// TwinCAT 3 PLC project TcCommando
// Title: TcCommando
// Company: Loupe
// Author: Loupe
// ProjectVersion: 0.0.1
// ProgramVersion: 3.1.4024.0
// libraries:
//   Tc2_Standard, * (Beckhoff Automation GmbH)
//   Tc2_System, * (Beckhoff Automation GmbH)
//   Tc3_Module, * (Beckhoff Automation GmbH)
//   TcPluginFramework, * (Loupe)
// project tree:
//   PLCOpen/DUT/ PLCOpenCallInternal.TcDUT, PLCOpenCallState.TcTLEO, PLCOpenCommandInternal.TcDUT (not stored), PLCOpenStatusBase.TcTLEO (not stored)
//   PLCOpen/Interfaces/ IPLCOpenBase.TcIO (not stored), IPLCOpenCall.TcIO, IPLCOpenCommand.TcIO (not stored), IPLCOpenGroup.TcIO
//   PLCOpen/POU/ PLCOpenCall.TcPOU, PLCOpenCallGroup.TcPOU (not stored), PLCOpenCallGroupType.TcDUT, PLCOpenCommand.TcPOU (not stored), PLCOpenCommandGroup.TcPOU, PLCOpenNullRemote.TcPOU (not stored)
//   / PlcTask.TcTTO
//   POUs/ MAIN.TcPOU (not stored)
// real-time tasks:
//   TASK PlcTask: cycle T#10ms, priority 20, ADS port 350

CONFIGURATION TcCommando
    RESOURCE PLC ON TwinCAT3
        TASK PlcTask(INTERVAL := T#10ms, PRIORITY := 20);
        PROGRAM MAIN WITH PlcTask : MAIN;
    END_RESOURCE
END_CONFIGURATION

// ---- PLCOpen/DUT/PLCOpenCallInternal.TcDUT
TYPE PLCOpenCallInternal :
STRUCT
	_state : PLCOpenCallState;
	_Command: IPLCOpenCommand;
	_abort: BOOL;
	_execute: BOOL;
	_break:BOOL;
	_RemoteStatus: PLCOPENSTATUSBASE;
	_self :IPLCOpenCall;
END_STRUCT
END_TYPE

// ---- PLCOpen/DUT/PLCOpenCallState.TcTLEO
{attribute 'qualified_only'}
{attribute 'strict'}
TYPE PLCOpenCallState :
(
	ATN_PLCOPEN_FUB_IDLE := 0,
	ATN_PLCOPEN_FUB_NEW_COMMAND,
	ATN_PLCOPEN_FUB_ABORTED,
	ATN_PLCOPEN_FUB_ABORT_OLD,
	ATN_PLCOPEN_FUB_STATUS,
	ATN_PLCOPEN_FUB_WRITE_PAR,
	ATN_PLCOPEN_FUB_SET_COMMAND,
	ATN_PLCOPEN_FUB_WORKING,
	ATN_PLCOPEN_FUB_CLEANUP,
	ATN_PLCOPEN_FUB_DONE
);
END_TYPE

// ---- PLCOpen/POU/PLCOpenCallGroupType.TcDUT
TYPE PLCOpenCallGroupType :
STRUCT
	_startStep : ENUM;  //The step when doStep was called
	_currentStep :ENUM;
	_lastRequestNumber : DINT;
	_onEntry : BOOL;
	_onExit : BOOL;
	_isDone : BOOL;
	_isAbort : BOOL;
	_isError : BOOL;
	_statusChecked : BOOL;
	_numberActiveCommands : INT;
	_commands : ARRAY[0..19] OF PLCOpenCall;
	_syncAbort : BOOL;
	_syncError : BOOL;
	_syncDone : BOOL;
END_STRUCT
END_TYPE

// ---- PLCOpen/Interfaces/IPLCOpenCall.TcIO
INTERFACE IPLCOpenCall

METHOD Aborted : BOOL
VAR_INPUT
END_VAR
END_METHOD

METHOD Errored : BOOL
VAR_INPUT
	ID : INT;
END_VAR
END_METHOD

METHOD Finished : BOOL
VAR_INPUT
END_VAR
END_METHOD

METHOD Start : BOOL
VAR_INPUT
	Command : IPLCOpenCommand;	
END_VAR
END_METHOD

END_INTERFACE

// ---- PLCOpen/Interfaces/IPLCOpenGroup.TcIO
INTERFACE IPLCOpenGroup

METHOD AbortPreviousCommands : BOOL
VAR_INPUT
	newCommand : IPLCOpenCommand;
END_VAR
END_METHOD

END_INTERFACE

// ---- PLCOpen/POU/PLCOpenCall.TcPOU
FUNCTION_BLOCK PLCOpenCall IMPLEMENTS IPLCOpenCall 
VAR_INPUT
	Execute : BOOL;
	Command : IPLCOpenCommand;
	Fallback: PLCOPENSTATUSBASE;
END_VAR
VAR_OUTPUT
	Status: PLCOPENSTATUSBASE;
	Busy : BOOL;
	Done : BOOL;
	Error : BOOL;
	CommandAborted : BOOL;
END_VAR
VAR
	i_PLCOpenCallInternal : PLCOpenCallInternal;
END_VAR

Call();

METHOD Aborted : BOOL
i_PLCOpenCallInternal._abort := true;
END_METHOD

METHOD Call : BOOL
VAR
	_break : BOOL;
END_VAR
	//Capture edges
	IF NOT Execute THEN
		i_PLCOpenCallInternal._execute := FALSE;
	END_IF

	//Start a new command on edge
	IF( Execute AND NOT i_PLCOpenCallInternal._execute)THEN
		i_PLCOpenCallInternal._execute := TRUE;
		i_PLCOpenCallInternal._state := PLCOpenCallState.ATN_PLCOPEN_FUB_NEW_COMMAND;
	END_IF
	
	//If we get aborted, handle it
	IF( i_PLCOpenCallInternal._abort )THEN
		i_PLCOpenCallInternal._abort := 0;
		i_PLCOpenCallInternal._state := PLCOpenCallState.ATN_PLCOPEN_FUB_ABORTED;
	END_IF

	i_PLCOpenCallInternal._self := THIS^;
	
	//We use a while not break so that we can do multiple passes at the state machine to do as much as possible in a single call	
	_break := FALSE;
	WHILE _break = FALSE DO
		CASE ( i_PLCOpenCallInternal._state ) OF
			//IDLE
			PLCOpenCallState.ATN_PLCOPEN_FUB_IDLE:
				Status := PLCOpenStatusBase.NOT_ENABLED;
				Busy := FALSE;
				Done := FALSE;
				Error := FALSE;
				CommandAborted := FALSE;
				_break := TRUE;
				
			//Start a new command by getting it
			PLCOpenCallState.ATN_PLCOPEN_FUB_NEW_COMMAND:
				Status := PLCOpenStatusBase.BUSY;
				i_PLCOpenCallInternal._RemoteStatus := PLCOpenStatusBase.BUSY;
				Busy := TRUE;
				Done := FALSE;
				Error := FALSE;
				CommandAborted := FALSE;			

				//If we are the current command:
				//1. we don't care about feedback
				//2. we don't want ourselves to get the abort
				//so remove this fub before calling abort previous
				IF i_PLCOpenCallInternal._Command <> 0 THEN
					IF i_PLCOpenCallInternal._Command.Remote = i_PLCOpenCallInternal._self THEN
						i_PLCOpenCallInternal._Command.Remote := 0; 
					END_IF
				END_IF 

				//Get the new command
				i_PLCOpenCallInternal._command := Command;
	
				IF i_PLCOpenCallInternal._Command <> 0 THEN
					i_PLCOpenCallInternal._state := PLCOpenCallState.ATN_PLCOPEN_FUB_ABORT_OLD;
					//No break;
				ELSE
					i_PLCOpenCallInternal._state := PLCOpenCallState.ATN_PLCOPEN_FUB_WORKING;
					i_PLCOpenCallInternal._RemoteStatus := Fallback;				
					_break := TRUE;
				END_IF

				//No break;
			
			//Abort any commands that was active using the same PLCOpen state
			PLCOpenCallState.ATN_PLCOPEN_FUB_ABORT_OLD:
				//This will 
				i_PLCOpenCallInternal._Command.AbortPreviousCommands(i_PLCOpenCallInternal._Command);

				i_PLCOpenCallInternal._state := PLCOpenCallState.ATN_PLCOPEN_FUB_SET_COMMAND;
				//no break;
				
			//Start the command
			PLCOpenCallState.ATN_PLCOPEN_FUB_SET_COMMAND:
				i_PLCOpenCallInternal._Command.Execute := TRUE;			
				i_PLCOpenCallInternal._Command.Remote := THIS^;			
			
				Busy := TRUE;
				i_PLCOpenCallInternal._state := PLCOpenCallState.ATN_PLCOPEN_FUB_WORKING;
				// no break
	
			//Wait for the command to be finished
			PLCOpenCallState.ATN_PLCOPEN_FUB_WORKING:
				Busy := TRUE;
				//No Break
	
				IF( i_PLCOpenCallInternal._RemoteStatus <> PLCOpenStatusBase.BUSY AND i_PLCOpenCallInternal._RemoteStatus <> PLCOpenStatusBase.ENABLED_WAITING ) THEN
					Status := i_PLCOpenCallInternal._RemoteStatus;
					Busy := FALSE;
					IF( Status = 0 ) THEN
						Done := TRUE;
					
					ELSE
						Error := TRUE;		
					END_IF
					i_PLCOpenCallInternal._state := PLCOpenCallState.ATN_PLCOPEN_FUB_CLEANUP;
					//no break;
				ELSE 
					_break := TRUE;
				END_IF
			
			//cleanup
			PLCOpenCallState.ATN_PLCOPEN_FUB_CLEANUP:
				//Remove self from the source command
				IF i_PLCOpenCallInternal._Command <> 0 THEN
					i_PLCOpenCallInternal._Command.Remote := 0;			
					i_PLCOpenCallInternal._Command := 0;
				END_IF
					
				i_PLCOpenCallInternal._state := PLCOpenCallState.ATN_PLCOPEN_FUB_DONE;
				//Break to force at least 1 cycle with statuses
				_break := TRUE;

			//done
			PLCOpenCallState.ATN_PLCOPEN_FUB_DONE:
	
				IF( NOT Execute )THEN
					i_PLCOpenCallInternal._state := PLCOpenCallState.ATN_PLCOPEN_FUB_IDLE;
					Status := PLCOpenStatusBase.NOT_ENABLED;
					Busy := FALSE;
					Done := FALSE;
					Error := FALSE;
					CommandAborted := FALSE;				
				END_IF
				_break := TRUE;
	
			//aborted
			PLCOpenCallState.ATN_PLCOPEN_FUB_ABORTED:
				Status := PLCOpenStatusBase.ABORTED;
				Busy := FALSE;
				Done := FALSE;
				Error := FALSE;
				CommandAborted := TRUE;
				i_PLCOpenCallInternal._command := 0;
				i_PLCOpenCallInternal._state := PLCOpenCallState.ATN_PLCOPEN_FUB_DONE;
				_break := TRUE;
					
		END_CASE
	END_WHILE
END_METHOD

METHOD Clear : PLCOpenStatusBase
THIS^.Execute := FALSE;
THIS^.i_PLCOpenCallInternal._state := PLCOpenCallState.ATN_PLCOPEN_FUB_CLEANUP;
//One call to cleanup
THIS^.Call();
//Second call to clear
THIS^.Call();
END_METHOD

METHOD Errored : BOOL
VAR_INPUT
	ID : INT;
END_VAR
CASE ID OF
	//Any of these statuses are invalid to return as an error.
	//Override to error
	PLCOPENSTATUSBASE.BUSY,
	PLCOPENSTATUSBASE.ENABLED_WAITING,
	PLCOPENSTATUSBASE.ERR_OK:
		i_PLCOpenCallInternal._RemoteStatus := PLCOPENSTATUSBASE.ERROR;
ELSE
	//Any other status can be passed through
	i_PLCOpenCallInternal._RemoteStatus := ID;
END_CASE
END_METHOD

METHOD Exec : PLCOpenStatusBase
VAR_INPUT
	Command : IPLCOpenCommand;	
END_VAR
//Abort the previous command if it exists
IF THIS^.Command <> Command THEN
	Command.Execute := FALSE;
	THIS^.Call();
END_IF

THIS^.Command := Command;
THIS^.Execute := TRUE;
THIS^.Call();
Exec := THIS^.Status;
END_METHOD

METHOD Finished : BOOL
i_PLCOpenCallInternal._RemoteStatus := PLCOpenStatusBase.ERR_OK;
END_METHOD

METHOD Start : BOOL
VAR_INPUT
	Command : IPLCOpenCommand;	
END_VAR
THIS^.Exec(Command);
END_METHOD

END_FUNCTION_BLOCK

// ---- PLCOpen/POU/PLCOpenCommandGroup.TcPOU
{attribute 'call_after_init'}
FUNCTION_BLOCK PLCOpenCommandGroup IMPLEMENTS IPLCOpenGroup
VAR_INPUT
	commands : ARRAY[0..19] OF  IPLCOpenCommand;
END_VAR

METHOD AbortPreviousCommands : BOOL
VAR_INPUT
	newCommand : IPLCOpenCommand;
END_VAR

VAR
	i: INT;
END_VAR
FOR i:=0 TO 19 DO

	IF commands[i] <> 0 AND commands[i] <> newCommand THEN

		commands[i].Aborted();

	END_IF	

END_FOR
END_METHOD

{attribute 'call_after_init'}
METHOD registerCommands : BOOL
VAR
	i : INT;
END_VAR
ADSLOGSTR(
	msgCtrlMask := ADSLOG_MSGTYPE_ERROR, 
	msgFmtStr   := 'Initing command group', 
	strArg      := '');  

FOR i:=0 TO 19 DO
	
	IF commands[i] <> 0 THEN

		commands[i].registerGroup(THIS^);
	
	END_IF
	
END_FOR
END_METHOD

END_FUNCTION_BLOCK
